(*********************************** G.D S.p.A. - Technical Department ***********************************
============= PROGRAM INFO ============
FOLDER:             TBD
MACHINES INVOLVED:  TBD 

============= DESCRIPTION =============
CSP: low task

============= REVISIONS ===============
Date		Version	 	Author      	Description             
----------	-------		------------  	--------------------------------------------
2019/04/05 	0000.00	 	G.Cera 			Creation of the PRG

**********************************************************************************************************)

PROGRAM _csp_low
VAR
END_VAR

_csp_case_low();

_csp_transfer_low();

_csp_main_low();

_csp_customerInterfaces_low();

END_PROGRAM

(* stored: Version 1.1.0.1, ProductVersion 3.1.4024.3
   POU _csp_low: Id {44c83cda-d58b-4c2d-a3d4-3abd21cccfd6}, SpecialFunc None *)
